Fanuc TP program (LS listing): MAKRO346.LS

/PROG  MAKRO346
/ATTR
OWNER		= MNEDITOR;
COMMENT		= "SPANNG.3_AUF/ZU";
PROG_SIZE	= 360;
CREATE		= DATE 10-09-17  TIME 16:56:34;
MODIFIED	= DATE 17-04-01  TIME 00:06:54;
FILE_NAME	= ;
VERSION		= 0;
LINE_COUNT	= 10;
MEMORY_SIZE	= 692;
PROTECT		= READ_WRITE;
TCD:  STACK_SIZE	= 0,
      TASK_PRIORITY	= 50,
      TIME_SLICE	= 0,
      BUSY_LAMP_OFF	= 0,
      ABORT_REQUEST	= 0,
      PAUSE_REQUEST	= 0;
DEFAULT_GROUP	= *,*,*,*,*;
CONTROL_CODE	= 00000000 00000000;
/MN
    :  !Spanngruppe 3 ZU/AUF ;
    :  !KS24 ;
    :  !Version: 01 ;
    :  !Stand: 001 ;
    :  !letzte  Aenderung  06.02.2015 LZ ;
    :  !Spanngruppe ZU ;
    :  DO[583]=(!F[23]) ;
    :  !Spanngruppe AUF ;
    :  DO[584]=(F[23]) ;
    :  F[26]=(ON) ;
/POS
/END
